(* Logix 5000 project; controller STAT 1756-L72 rev 20.12; software revision 20.04; part 27 of 34 *)
(* tags used below, declared in another part *)
   B3 : DINT[35];
   N20 : DINT[50];
   N7 : DINT[150];
   N9 : DINT[200];
   S : INT[164];
   T4 : TIMER[100];
   S_ppas_HT : DINT;
   S_ppas_l1op008 : DINT;
   S_ppas_L2op008 : DINT;
(* LANCY, continued *)

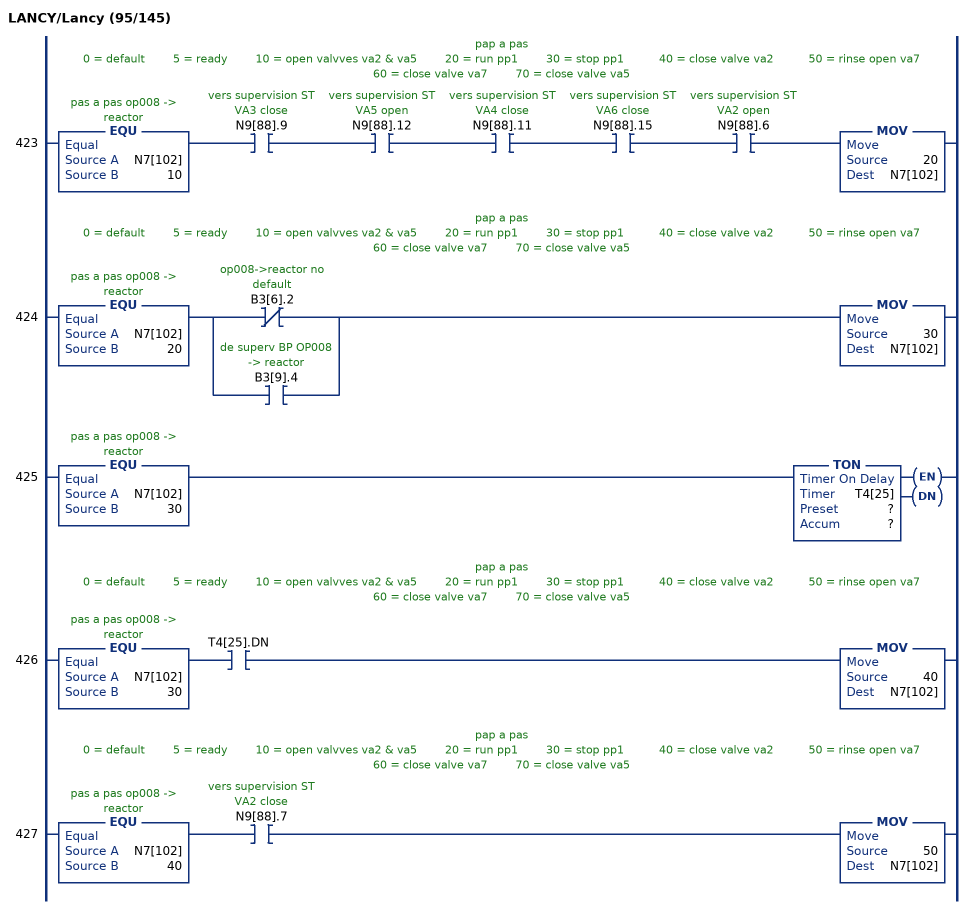
   // pap a pas
   // 0 = default        5 = ready        10 = open valvves va2 & va5        20 = run pp1        30 = stop pp1          40 = close valve va2          50 = rinse open va7            60 = close valve va7        70 = close valve va5
   423: EQU(N7[102],10)XIC(N9[88].9)XIC(N9[88].12)XIC(N9[88].11)XIC(N9[88].15)XIC(N9[88].6)MOV(20,N7[102]);
   // pap a pas
   // 0 = default        5 = ready        10 = open valvves va2 & va5        20 = run pp1        30 = stop pp1          40 = close valve va2          50 = rinse open va7            60 = close valve va7        70 = close valve va5
   424: EQU(N7[102],20)[XIO(B3[6].2) ,XIC(B3[9].4) ]MOV(30,N7[102]);
   425: EQU(N7[102],30)TON(T4[25],?,?);
   // pap a pas
   // 0 = default        5 = ready        10 = open valvves va2 & va5        20 = run pp1        30 = stop pp1          40 = close valve va2          50 = rinse open va7            60 = close valve va7        70 = close valve va5
   426: EQU(N7[102],30)XIC(T4[25].DN)MOV(40,N7[102]);
   // pap a pas
   // 0 = default        5 = ready        10 = open valvves va2 & va5        20 = run pp1        30 = stop pp1          40 = close valve va2          50 = rinse open va7            60 = close valve va7        70 = close valve va5
   427: EQU(N7[102],40)XIC(N9[88].7)MOV(50,N7[102]);
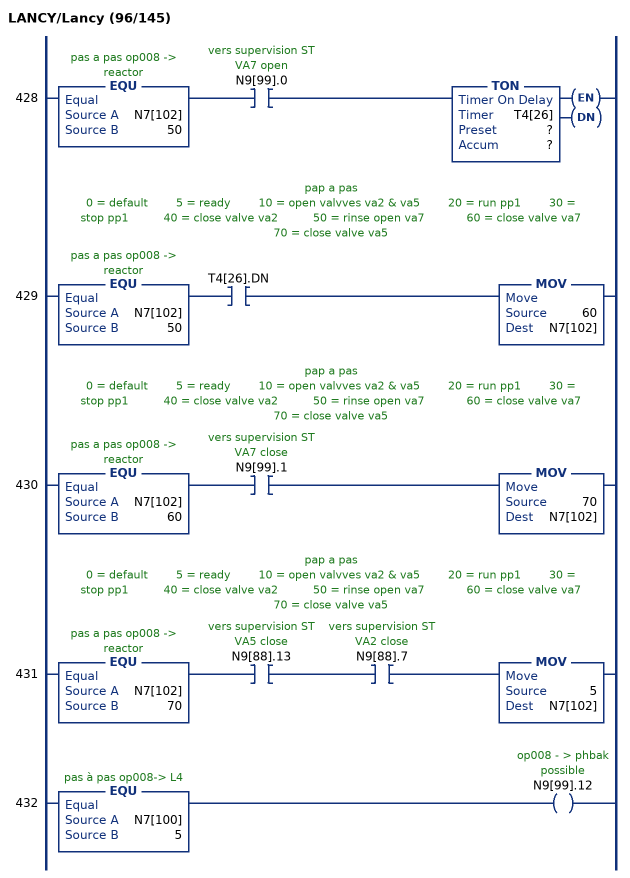
   428: EQU(N7[102],50)XIC(N9[99].0)TON(T4[26],?,?);
   // pap a pas
   // 0 = default        5 = ready        10 = open valvves va2 & va5        20 = run pp1        30 = stop pp1          40 = close valve va2          50 = rinse open va7            60 = close valve va7        70 = close valve va5
   429: EQU(N7[102],50)XIC(T4[26].DN)MOV(60,N7[102]);
   // pap a pas
   // 0 = default        5 = ready        10 = open valvves va2 & va5        20 = run pp1        30 = stop pp1          40 = close valve va2          50 = rinse open va7            60 = close valve va7        70 = close valve va5
   430: EQU(N7[102],60)XIC(N9[99].1)MOV(70,N7[102]);
   // pap a pas
   // 0 = default        5 = ready        10 = open valvves va2 & va5        20 = run pp1        30 = stop pp1          40 = close valve va2          50 = rinse open va7            60 = close valve va7        70 = close valve va5
   431: EQU(N7[102],70)XIC(N9[88].13)XIC(N9[88].7)MOV(5,N7[102]);
   432: EQU(N7[100],5)OTE(N9[99].12);
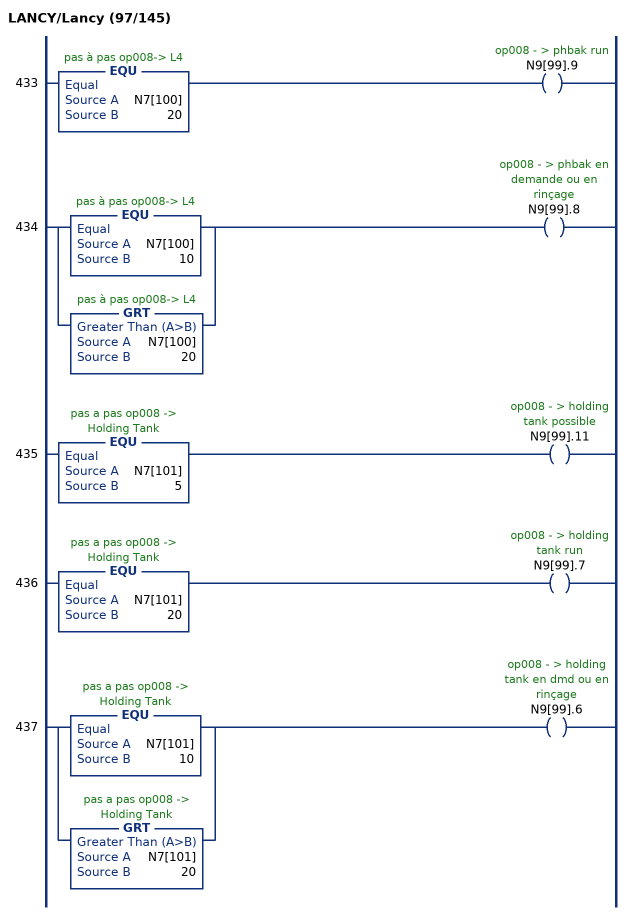
   433: EQU(N7[100],20)OTE(N9[99].9);
   434: [EQU(N7[100],10) ,GRT(N7[100],20) ]OTE(N9[99].8);
   435: EQU(N7[101],5)OTE(N9[99].11);
   436: EQU(N7[101],20)OTE(N9[99].7);
   437: [EQU(N7[101],10) ,GRT(N7[101],20) ]OTE(N9[99].6);
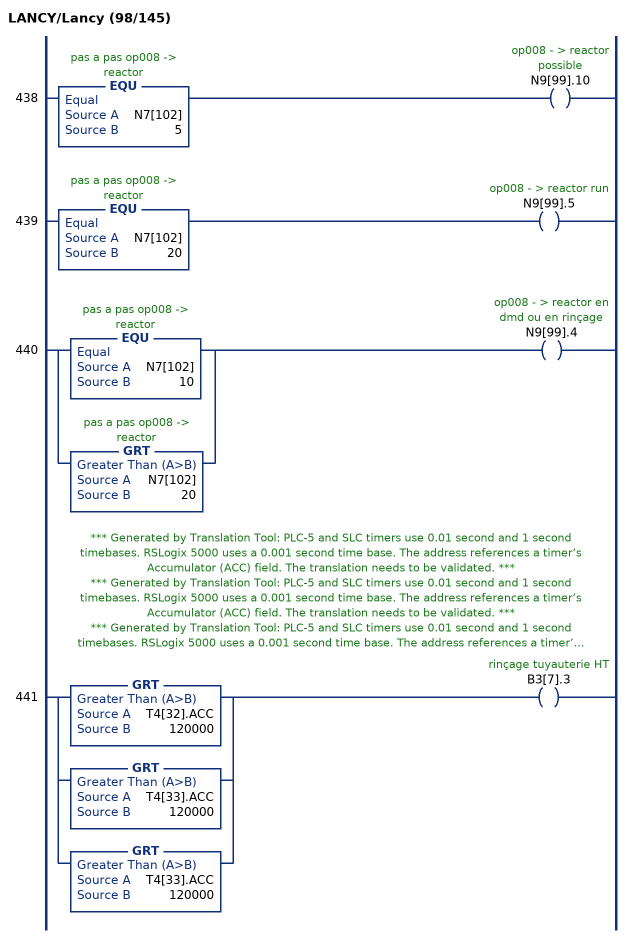
   438: EQU(N7[102],5)OTE(N9[99].10);
   439: EQU(N7[102],20)OTE(N9[99].5);
   440: [EQU(N7[102],10) ,GRT(N7[102],20) ]OTE(N9[99].4);
   // *** Generated by Translation Tool: PLC-5 and SLC timers use 0.01 second and 1 second timebases. RSLogix 5000 uses a 0.001 second time base. The address references a timer’s Accumulator (ACC) field. The translation needs to be validated. ***
   // *** Generated by Translation Tool: PLC-5 and SLC timers use 0.01 second and 1 second timebases. RSLogix 5000 uses a 0.001 second time base. The address references a timer’s Accumulator (ACC) field. The translation needs to be validated. ***
   // *** Generated by Translation Tool: PLC-5 and SLC timers use 0.01 second and 1 second timebases. RSLogix 5000 uses a 0.001 second time base. The address references a timer’s Accumulator (ACC) field. The translation needs to be validated. ***
   441: [GRT(T4[32].ACC,120000) ,GRT(T4[33].ACC,120000) ,GRT(T4[33].ACC,120000) ]OTE(B3[7].3);
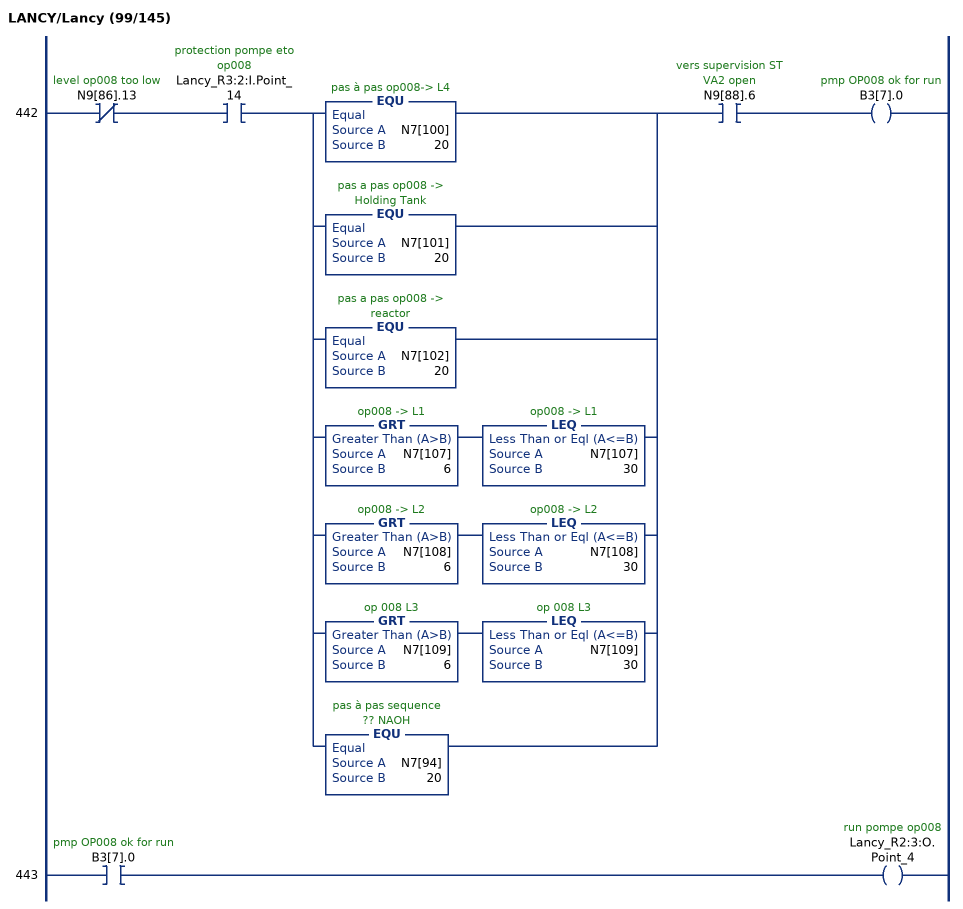
   442: XIO(N9[86].13)XIC(Lancy_R3:2:I.Point_14)[EQU(N7[100],20) ,EQU(N7[101],20) ,EQU(N7[102],20) ,GRT(N7[107],6) LEQ(N7[107],30) ,GRT(N7[108],6) LEQ(N7[108],30) ,GRT(N7[109],6) LEQ(N7[109],30) ,EQU(N7[94],20) ]XIC(N9[88].6)OTE(B3[7].0);
   443: XIC(B3[7].0)OTE(Lancy_R2:3:O.Point_4);
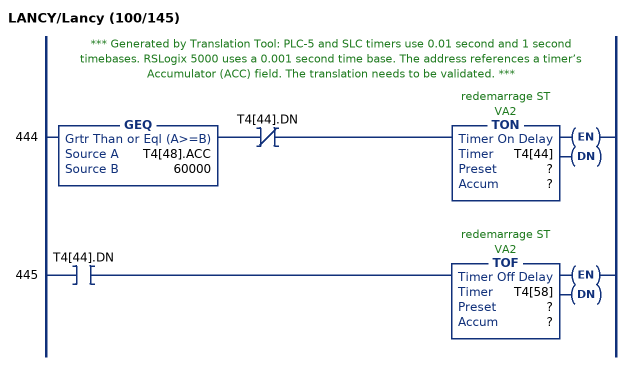
   // *** Generated by Translation Tool: PLC-5 and SLC timers use 0.01 second and 1 second timebases. RSLogix 5000 uses a 0.001 second time base. The address references a timer’s Accumulator (ACC) field. The translation needs to be validated. ***
   444: GEQ(T4[48].ACC,60000)XIO(T4[44].DN)TON(T4[44],?,?);
   445: XIC(T4[44].DN)TOF(T4[58],?,?);
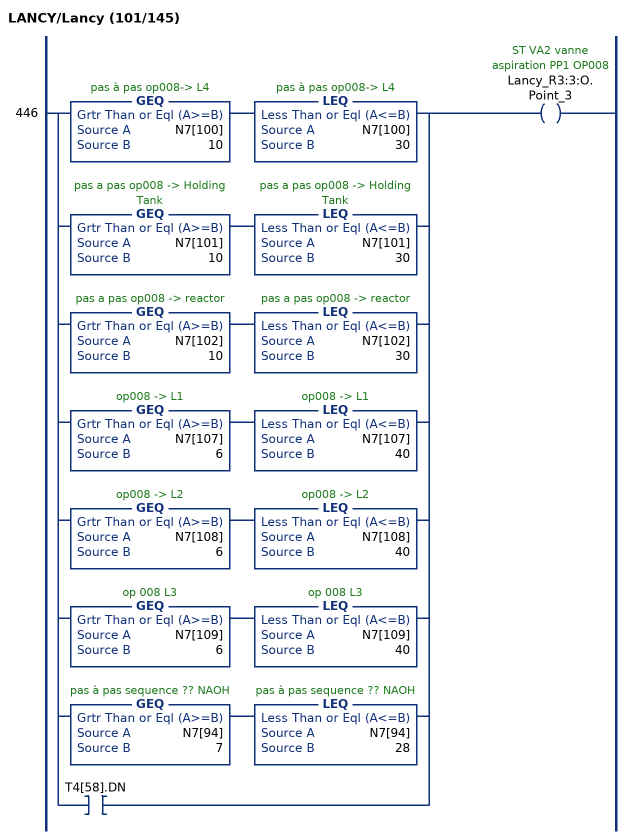
   446: [GEQ(N7[100],10) LEQ(N7[100],30) ,GEQ(N7[101],10) LEQ(N7[101],30) ,GEQ(N7[102],10) LEQ(N7[102],30) ,GEQ(N7[107],6) LEQ(N7[107],40) ,GEQ(N7[108],6) LEQ(N7[108],40) ,GEQ(N7[109],6) LEQ(N7[109],40) ,GEQ(N7[94],7) LEQ(N7[94],28) ,XIC(T4[58].DN) ]OTE(Lancy_R3:3:O.Point_3);
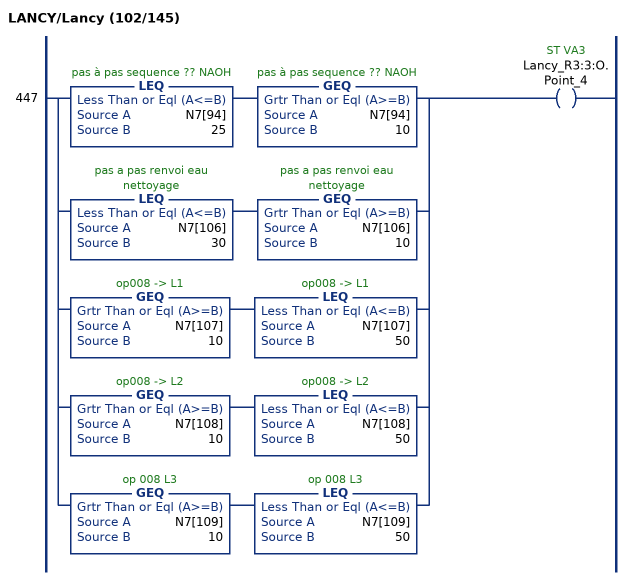
   447: [LEQ(N7[94],25) GEQ(N7[94],10) ,LEQ(N7[106],30) GEQ(N7[106],10) ,GEQ(N7[107],10) LEQ(N7[107],50) ,GEQ(N7[108],10) LEQ(N7[108],50) ,GEQ(N7[109],10) LEQ(N7[109],50) ]OTE(Lancy_R3:3:O.Point_4);
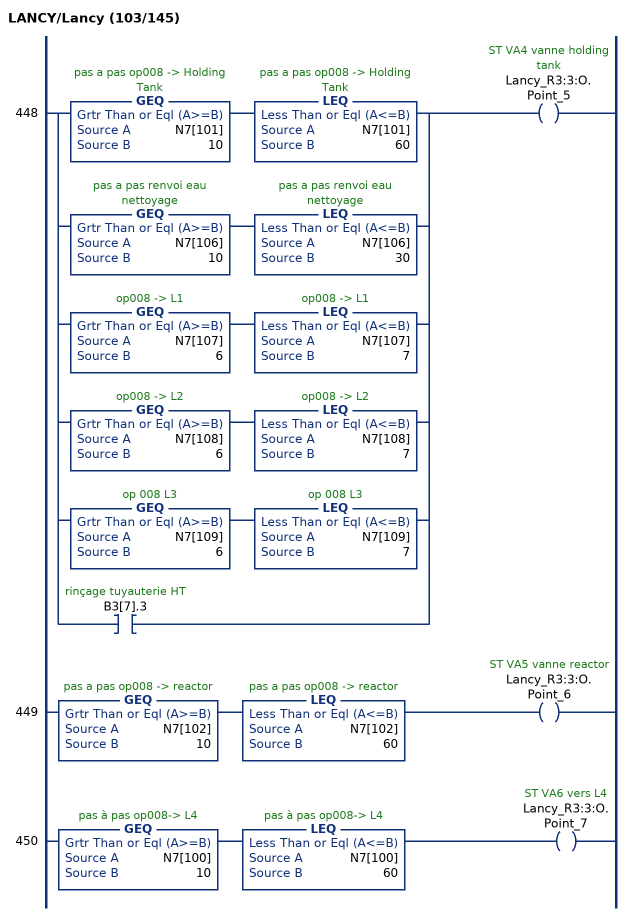
   448: [GEQ(N7[101],10) LEQ(N7[101],60) ,GEQ(N7[106],10) LEQ(N7[106],30) ,GEQ(N7[107],6) LEQ(N7[107],7) ,GEQ(N7[108],6) LEQ(N7[108],7) ,GEQ(N7[109],6) LEQ(N7[109],7) ,XIC(B3[7].3) ]OTE(Lancy_R3:3:O.Point_5);
   449: GEQ(N7[102],10)LEQ(N7[102],60)OTE(Lancy_R3:3:O.Point_6);
   450: GEQ(N7[100],10)LEQ(N7[100],60)OTE(Lancy_R3:3:O.Point_7);
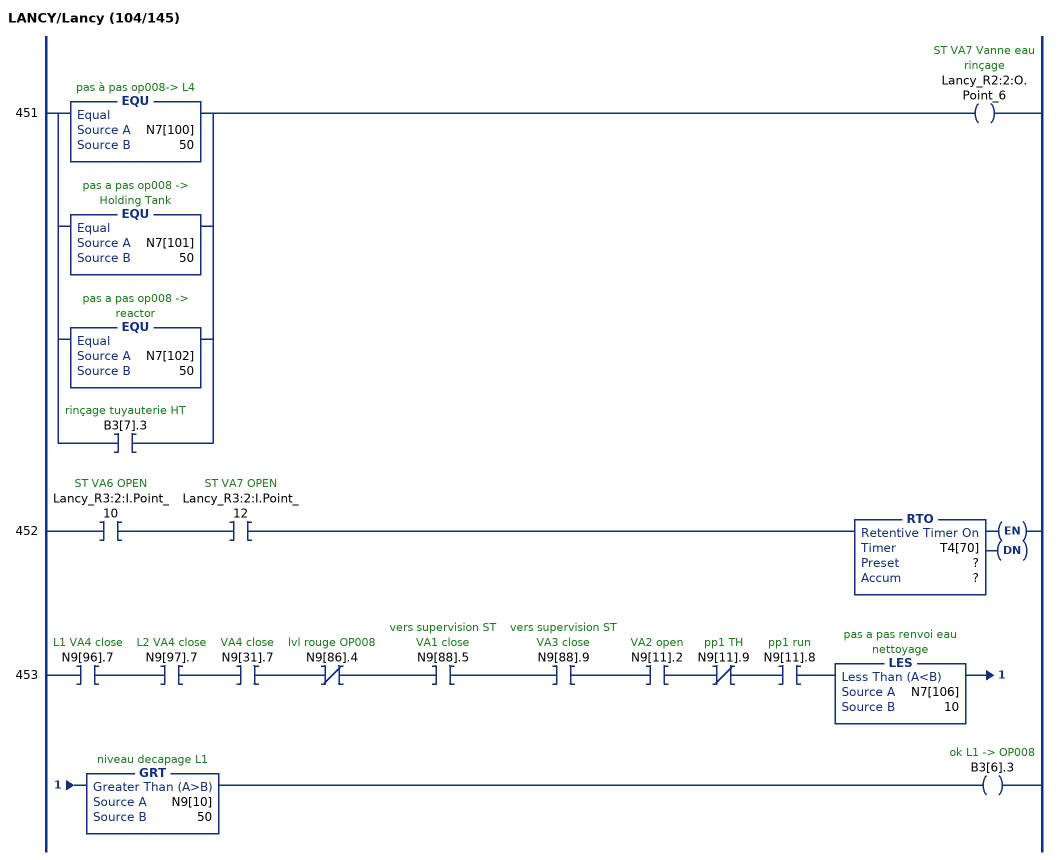
   451: [EQU(N7[100],50) ,EQU(N7[101],50) ,EQU(N7[102],50) ,XIC(B3[7].3) ]OTE(Lancy_R2:2:O.Point_6);
   452: XIC(Lancy_R3:2:I.Point_10)XIC(Lancy_R3:2:I.Point_12)RTO(T4[70],?,?);
   453: XIC(N9[96].7)XIC(N9[97].7)XIC(N9[31].7)XIO(N9[86].4)XIC(N9[88].5)XIC(N9[88].9)XIC(N9[11].2)XIO(N9[11].9)XIC(N9[11].8)LES(N7[106],10)GRT(N9[10],50)OTE(B3[6].3);
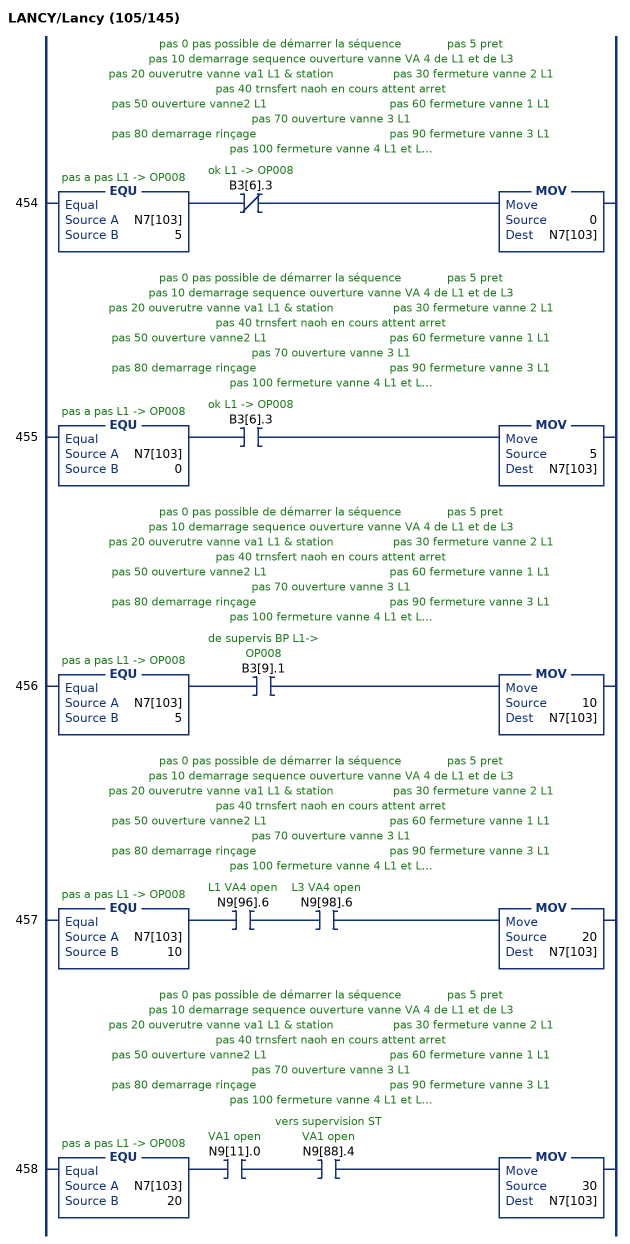
   // pas 0 pas possible de démarrer la séquence             pas 5 pret                                                 pas 10 demarrage sequence ouverture vanne VA 4 de L1 et de L3
   // pas 20 ouverutre vanne va1 L1 & station                 pas 30 fermeture vanne 2 L1                       pas 40 trnsfert naoh en cours attent arret
   // pas 50 ouverture vanne2 L1                                   pas 60 fermeture vanne 1 L1                       pas 70 ouverture vanne 3 L1
   // pas 80 demarrage rinçage                                      pas 90 fermeture vanne 3 L1                       pas 100 fermeture vanne 4 L1 et L3
   // pas 110 fermeture vanne station 1
   454: EQU(N7[103],5)XIO(B3[6].3)MOV(0,N7[103]);
   // pas 0 pas possible de démarrer la séquence             pas 5 pret                                                 pas 10 demarrage sequence ouverture vanne VA 4 de L1 et de L3
   // pas 20 ouverutre vanne va1 L1 & station                 pas 30 fermeture vanne 2 L1                       pas 40 trnsfert naoh en cours attent arret
   // pas 50 ouverture vanne2 L1                                   pas 60 fermeture vanne 1 L1                       pas 70 ouverture vanne 3 L1
   // pas 80 demarrage rinçage                                      pas 90 fermeture vanne 3 L1                       pas 100 fermeture vanne 4 L1 et L3
   // pas 110 fermeture vanne station 1
   455: EQU(N7[103],0)XIC(B3[6].3)MOV(5,N7[103]);
   // pas 0 pas possible de démarrer la séquence             pas 5 pret                                                 pas 10 demarrage sequence ouverture vanne VA 4 de L1 et de L3
   // pas 20 ouverutre vanne va1 L1 & station                 pas 30 fermeture vanne 2 L1                       pas 40 trnsfert naoh en cours attent arret
   // pas 50 ouverture vanne2 L1                                   pas 60 fermeture vanne 1 L1                       pas 70 ouverture vanne 3 L1
   // pas 80 demarrage rinçage                                      pas 90 fermeture vanne 3 L1                       pas 100 fermeture vanne 4 L1 et L3
   // pas 110 fermeture vanne station 1
   456: EQU(N7[103],5)XIC(B3[9].1)MOV(10,N7[103]);
   // pas 0 pas possible de démarrer la séquence             pas 5 pret                                                 pas 10 demarrage sequence ouverture vanne VA 4 de L1 et de L3
   // pas 20 ouverutre vanne va1 L1 & station                 pas 30 fermeture vanne 2 L1                       pas 40 trnsfert naoh en cours attent arret
   // pas 50 ouverture vanne2 L1                                   pas 60 fermeture vanne 1 L1                       pas 70 ouverture vanne 3 L1
   // pas 80 demarrage rinçage                                      pas 90 fermeture vanne 3 L1                       pas 100 fermeture vanne 4 L1 et L3
   // pas 110 fermeture vanne station 1
   457: EQU(N7[103],10)XIC(N9[96].6)XIC(N9[98].6)MOV(20,N7[103]);
   // pas 0 pas possible de démarrer la séquence             pas 5 pret                                                 pas 10 demarrage sequence ouverture vanne VA 4 de L1 et de L3
   // pas 20 ouverutre vanne va1 L1 & station                 pas 30 fermeture vanne 2 L1                       pas 40 trnsfert naoh en cours attent arret
   // pas 50 ouverture vanne2 L1                                   pas 60 fermeture vanne 1 L1                       pas 70 ouverture vanne 3 L1
   // pas 80 demarrage rinçage                                      pas 90 fermeture vanne 3 L1                       pas 100 fermeture vanne 4 L1 et L3
   // pas 110 fermeture vanne station 1
   458: EQU(N7[103],20)XIC(N9[11].0)XIC(N9[88].4)MOV(30,N7[103]);
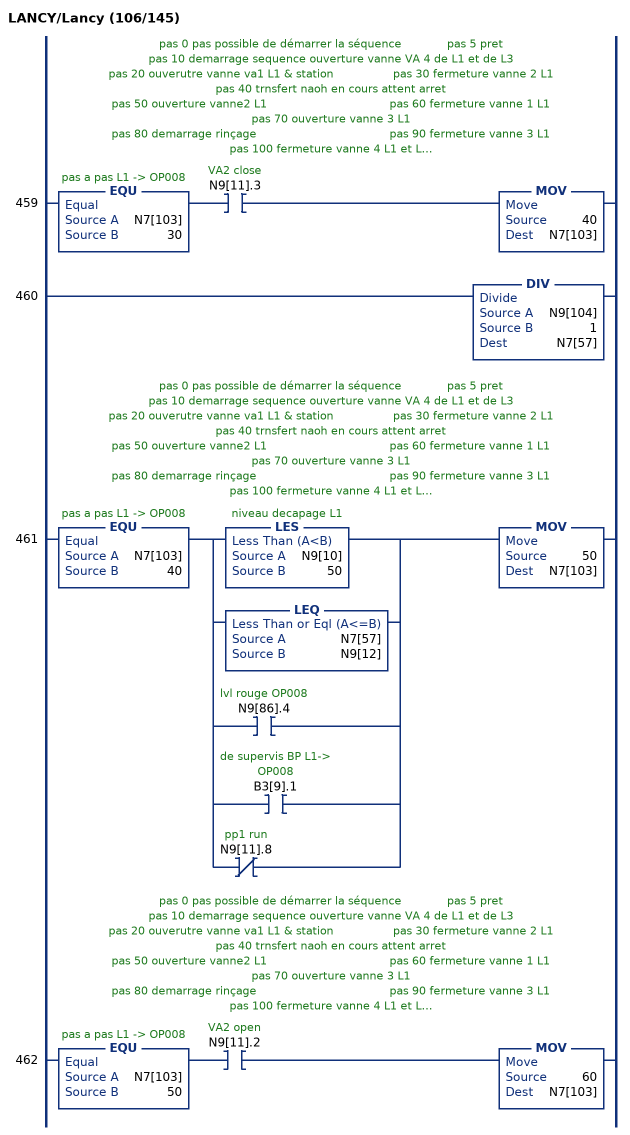
   // pas 0 pas possible de démarrer la séquence             pas 5 pret                                                 pas 10 demarrage sequence ouverture vanne VA 4 de L1 et de L3
   // pas 20 ouverutre vanne va1 L1 & station                 pas 30 fermeture vanne 2 L1                       pas 40 trnsfert naoh en cours attent arret
   // pas 50 ouverture vanne2 L1                                   pas 60 fermeture vanne 1 L1                       pas 70 ouverture vanne 3 L1
   // pas 80 demarrage rinçage                                      pas 90 fermeture vanne 3 L1                       pas 100 fermeture vanne 4 L1 et L3
   // pas 110 fermeture vanne station 1
   459: EQU(N7[103],30)XIC(N9[11].3)MOV(40,N7[103]);
   460: DIV(N9[104],1,N7[57]);
   // pas 0 pas possible de démarrer la séquence             pas 5 pret                                                 pas 10 demarrage sequence ouverture vanne VA 4 de L1 et de L3
   // pas 20 ouverutre vanne va1 L1 & station                 pas 30 fermeture vanne 2 L1                       pas 40 trnsfert naoh en cours attent arret
   // pas 50 ouverture vanne2 L1                                   pas 60 fermeture vanne 1 L1                       pas 70 ouverture vanne 3 L1
   // pas 80 demarrage rinçage                                      pas 90 fermeture vanne 3 L1                       pas 100 fermeture vanne 4 L1 et L3
   // pas 110 fermeture vanne station 1
   461: EQU(N7[103],40)[LES(N9[10],50) ,LEQ(N7[57],N9[12]) ,XIC(N9[86].4) ,XIC(B3[9].1) ,XIO(N9[11].8) ]MOV(50,N7[103]);
   // pas 0 pas possible de démarrer la séquence             pas 5 pret                                                 pas 10 demarrage sequence ouverture vanne VA 4 de L1 et de L3
   // pas 20 ouverutre vanne va1 L1 & station                 pas 30 fermeture vanne 2 L1                       pas 40 trnsfert naoh en cours attent arret
   // pas 50 ouverture vanne2 L1                                   pas 60 fermeture vanne 1 L1                       pas 70 ouverture vanne 3 L1
   // pas 80 demarrage rinçage                                      pas 90 fermeture vanne 3 L1                       pas 100 fermeture vanne 4 L1 et L3
   // pas 110 fermeture vanne station 1
   462: EQU(N7[103],50)XIC(N9[11].2)MOV(60,N7[103]);
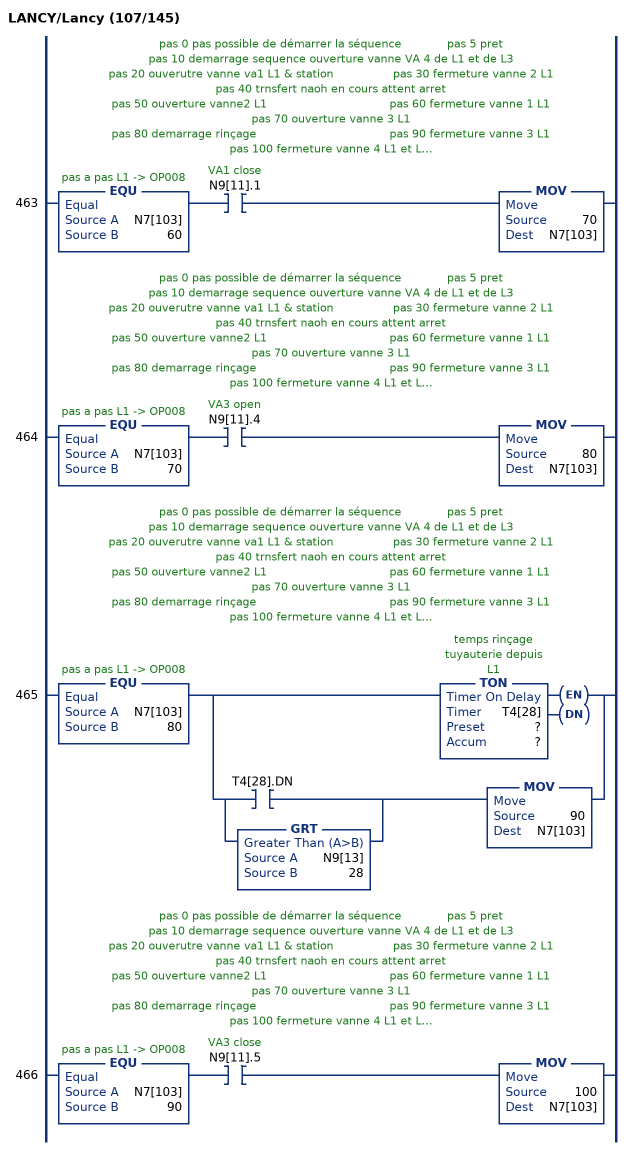
   // pas 0 pas possible de démarrer la séquence             pas 5 pret                                                 pas 10 demarrage sequence ouverture vanne VA 4 de L1 et de L3
   // pas 20 ouverutre vanne va1 L1 & station                 pas 30 fermeture vanne 2 L1                       pas 40 trnsfert naoh en cours attent arret
   // pas 50 ouverture vanne2 L1                                   pas 60 fermeture vanne 1 L1                       pas 70 ouverture vanne 3 L1
   // pas 80 demarrage rinçage                                      pas 90 fermeture vanne 3 L1                       pas 100 fermeture vanne 4 L1 et L3
   // pas 110 fermeture vanne station 1
   463: EQU(N7[103],60)XIC(N9[11].1)MOV(70,N7[103]);
   // pas 0 pas possible de démarrer la séquence             pas 5 pret                                                 pas 10 demarrage sequence ouverture vanne VA 4 de L1 et de L3
   // pas 20 ouverutre vanne va1 L1 & station                 pas 30 fermeture vanne 2 L1                       pas 40 trnsfert naoh en cours attent arret
   // pas 50 ouverture vanne2 L1                                   pas 60 fermeture vanne 1 L1                       pas 70 ouverture vanne 3 L1
   // pas 80 demarrage rinçage                                      pas 90 fermeture vanne 3 L1                       pas 100 fermeture vanne 4 L1 et L3
   // pas 110 fermeture vanne station 1
   464: EQU(N7[103],70)XIC(N9[11].4)MOV(80,N7[103]);
   // pas 0 pas possible de démarrer la séquence             pas 5 pret                                                 pas 10 demarrage sequence ouverture vanne VA 4 de L1 et de L3
   // pas 20 ouverutre vanne va1 L1 & station                 pas 30 fermeture vanne 2 L1                       pas 40 trnsfert naoh en cours attent arret
   // pas 50 ouverture vanne2 L1                                   pas 60 fermeture vanne 1 L1                       pas 70 ouverture vanne 3 L1
   // pas 80 demarrage rinçage                                      pas 90 fermeture vanne 3 L1                       pas 100 fermeture vanne 4 L1 et L3
   // pas 110 fermeture vanne station 1
   465: EQU(N7[103],80)[TON(T4[28],?,?) ,[XIC(T4[28].DN) ,GRT(N9[13],28) ] MOV(90,N7[103]) ];
   // pas 0 pas possible de démarrer la séquence             pas 5 pret                                                 pas 10 demarrage sequence ouverture vanne VA 4 de L1 et de L3
   // pas 20 ouverutre vanne va1 L1 & station                 pas 30 fermeture vanne 2 L1                       pas 40 trnsfert naoh en cours attent arret
   // pas 50 ouverture vanne2 L1                                   pas 60 fermeture vanne 1 L1                       pas 70 ouverture vanne 3 L1
   // pas 80 demarrage rinçage                                      pas 90 fermeture vanne 3 L1                       pas 100 fermeture vanne 4 L1 et L3
   // pas 110 fermeture vanne station 1
   466: EQU(N7[103],90)XIC(N9[11].5)MOV(100,N7[103]);
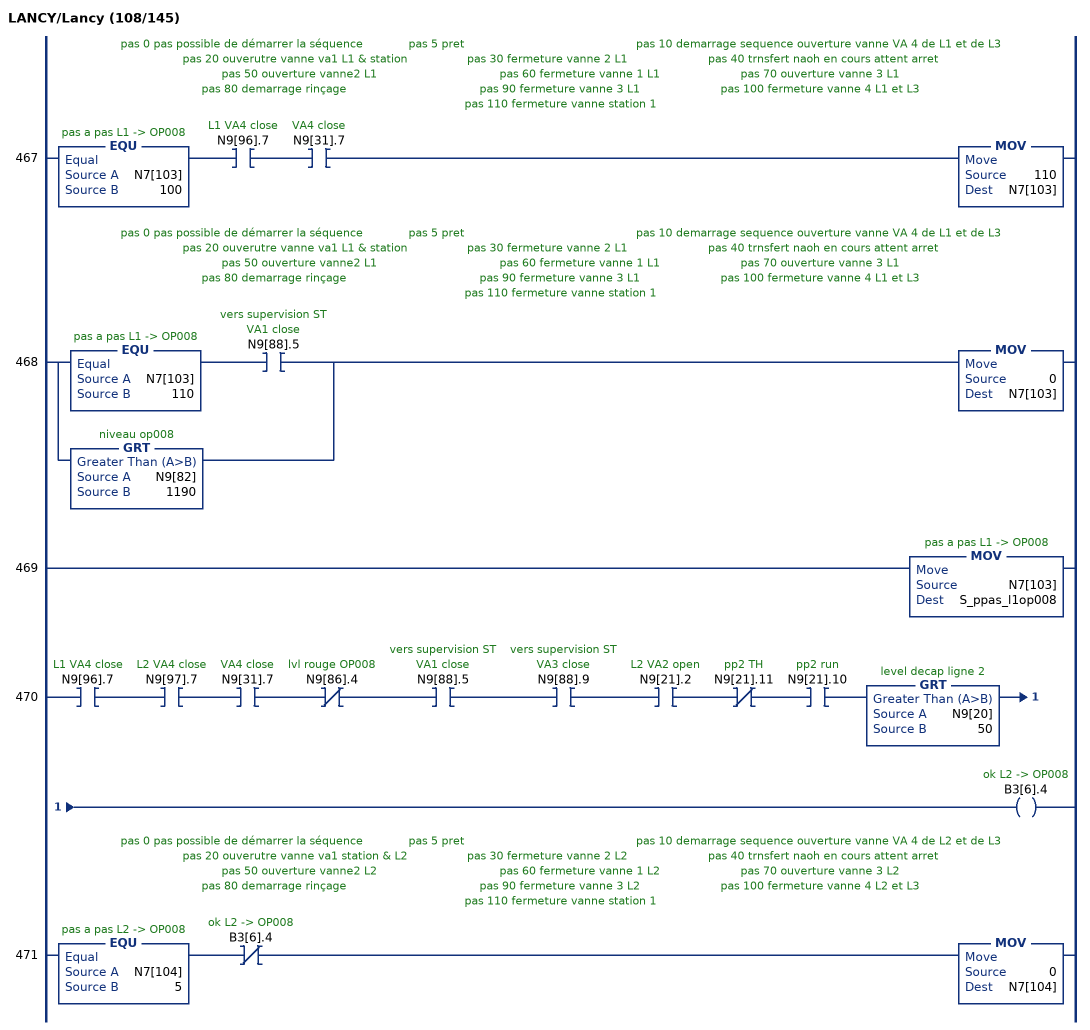
   // pas 0 pas possible de démarrer la séquence             pas 5 pret                                                 pas 10 demarrage sequence ouverture vanne VA 4 de L1 et de L3
   // pas 20 ouverutre vanne va1 L1 & station                 pas 30 fermeture vanne 2 L1                       pas 40 trnsfert naoh en cours attent arret
   // pas 50 ouverture vanne2 L1                                   pas 60 fermeture vanne 1 L1                       pas 70 ouverture vanne 3 L1
   // pas 80 demarrage rinçage                                      pas 90 fermeture vanne 3 L1                       pas 100 fermeture vanne 4 L1 et L3
   // pas 110 fermeture vanne station 1
   467: EQU(N7[103],100)XIC(N9[96].7)XIC(N9[31].7)MOV(110,N7[103]);
   // pas 0 pas possible de démarrer la séquence             pas 5 pret                                                 pas 10 demarrage sequence ouverture vanne VA 4 de L1 et de L3
   // pas 20 ouverutre vanne va1 L1 & station                 pas 30 fermeture vanne 2 L1                       pas 40 trnsfert naoh en cours attent arret
   // pas 50 ouverture vanne2 L1                                   pas 60 fermeture vanne 1 L1                       pas 70 ouverture vanne 3 L1
   // pas 80 demarrage rinçage                                      pas 90 fermeture vanne 3 L1                       pas 100 fermeture vanne 4 L1 et L3
   // pas 110 fermeture vanne station 1
   468: [EQU(N7[103],110) XIC(N9[88].5) ,GRT(N9[82],1190) ]MOV(0,N7[103]);
   469: MOV(N7[103],S_ppas_l1op008);
   470: XIC(N9[96].7)XIC(N9[97].7)XIC(N9[31].7)XIO(N9[86].4)XIC(N9[88].5)XIC(N9[88].9)XIC(N9[21].2)XIO(N9[21].11)XIC(N9[21].10)GRT(N9[20],50)OTE(B3[6].4);
   // pas 0 pas possible de démarrer la séquence             pas 5 pret                                                 pas 10 demarrage sequence ouverture vanne VA 4 de L2 et de L3
   // pas 20 ouverutre vanne va1 station & L2                 pas 30 fermeture vanne 2 L2                       pas 40 trnsfert naoh en cours attent arret
   // pas 50 ouverture vanne2 L2                                   pas 60 fermeture vanne 1 L2                       pas 70 ouverture vanne 3 L2
   // pas 80 demarrage rinçage                                      pas 90 fermeture vanne 3 L2                       pas 100 fermeture vanne 4 L2 et L3
   // pas 110 fermeture vanne station 1
   471: EQU(N7[104],5)XIO(B3[6].4)MOV(0,N7[104]);
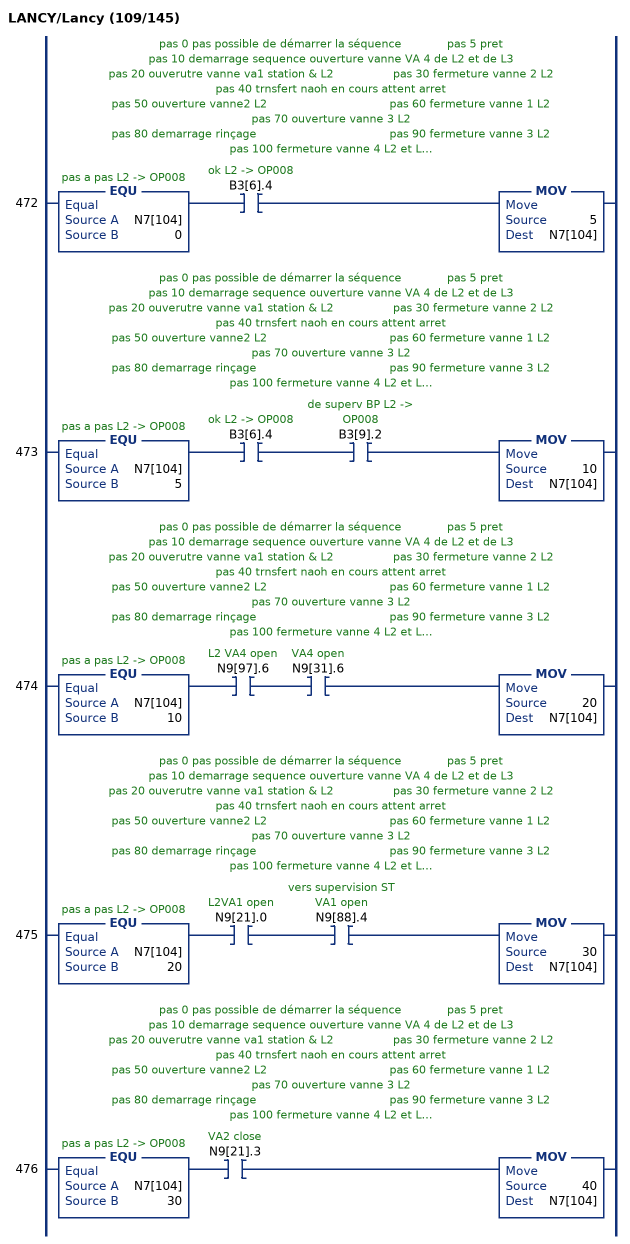
   // pas 0 pas possible de démarrer la séquence             pas 5 pret                                                 pas 10 demarrage sequence ouverture vanne VA 4 de L2 et de L3
   // pas 20 ouverutre vanne va1 station & L2                 pas 30 fermeture vanne 2 L2                       pas 40 trnsfert naoh en cours attent arret
   // pas 50 ouverture vanne2 L2                                   pas 60 fermeture vanne 1 L2                       pas 70 ouverture vanne 3 L2
   // pas 80 demarrage rinçage                                      pas 90 fermeture vanne 3 L2                       pas 100 fermeture vanne 4 L2 et L3
   // pas 110 fermeture vanne station 1
   472: EQU(N7[104],0)XIC(B3[6].4)MOV(5,N7[104]);
   // pas 0 pas possible de démarrer la séquence             pas 5 pret                                                 pas 10 demarrage sequence ouverture vanne VA 4 de L2 et de L3
   // pas 20 ouverutre vanne va1 station & L2                 pas 30 fermeture vanne 2 L2                       pas 40 trnsfert naoh en cours attent arret
   // pas 50 ouverture vanne2 L2                                   pas 60 fermeture vanne 1 L2                       pas 70 ouverture vanne 3 L2
   // pas 80 demarrage rinçage                                      pas 90 fermeture vanne 3 L2                       pas 100 fermeture vanne 4 L2 et L3
   // pas 110 fermeture vanne station 1
   473: EQU(N7[104],5)XIC(B3[6].4)XIC(B3[9].2)MOV(10,N7[104]);
   // pas 0 pas possible de démarrer la séquence             pas 5 pret                                                 pas 10 demarrage sequence ouverture vanne VA 4 de L2 et de L3
   // pas 20 ouverutre vanne va1 station & L2                 pas 30 fermeture vanne 2 L2                       pas 40 trnsfert naoh en cours attent arret
   // pas 50 ouverture vanne2 L2                                   pas 60 fermeture vanne 1 L2                       pas 70 ouverture vanne 3 L2
   // pas 80 demarrage rinçage                                      pas 90 fermeture vanne 3 L2                       pas 100 fermeture vanne 4 L2 et L3
   // pas 110 fermeture vanne station 1
   474: EQU(N7[104],10)XIC(N9[97].6)XIC(N9[31].6)MOV(20,N7[104]);
   // pas 0 pas possible de démarrer la séquence             pas 5 pret                                                 pas 10 demarrage sequence ouverture vanne VA 4 de L2 et de L3
   // pas 20 ouverutre vanne va1 station & L2                 pas 30 fermeture vanne 2 L2                       pas 40 trnsfert naoh en cours attent arret
   // pas 50 ouverture vanne2 L2                                   pas 60 fermeture vanne 1 L2                       pas 70 ouverture vanne 3 L2
   // pas 80 demarrage rinçage                                      pas 90 fermeture vanne 3 L2                       pas 100 fermeture vanne 4 L2 et L3
   // pas 110 fermeture vanne station 1
   475: EQU(N7[104],20)XIC(N9[21].0)XIC(N9[88].4)MOV(30,N7[104]);
   // pas 0 pas possible de démarrer la séquence             pas 5 pret                                                 pas 10 demarrage sequence ouverture vanne VA 4 de L2 et de L3
   // pas 20 ouverutre vanne va1 station & L2                 pas 30 fermeture vanne 2 L2                       pas 40 trnsfert naoh en cours attent arret
   // pas 50 ouverture vanne2 L2                                   pas 60 fermeture vanne 1 L2                       pas 70 ouverture vanne 3 L2
   // pas 80 demarrage rinçage                                      pas 90 fermeture vanne 3 L2                       pas 100 fermeture vanne 4 L2 et L3
   // pas 110 fermeture vanne station 1
   476: EQU(N7[104],30)XIC(N9[21].3)MOV(40,N7[104]);
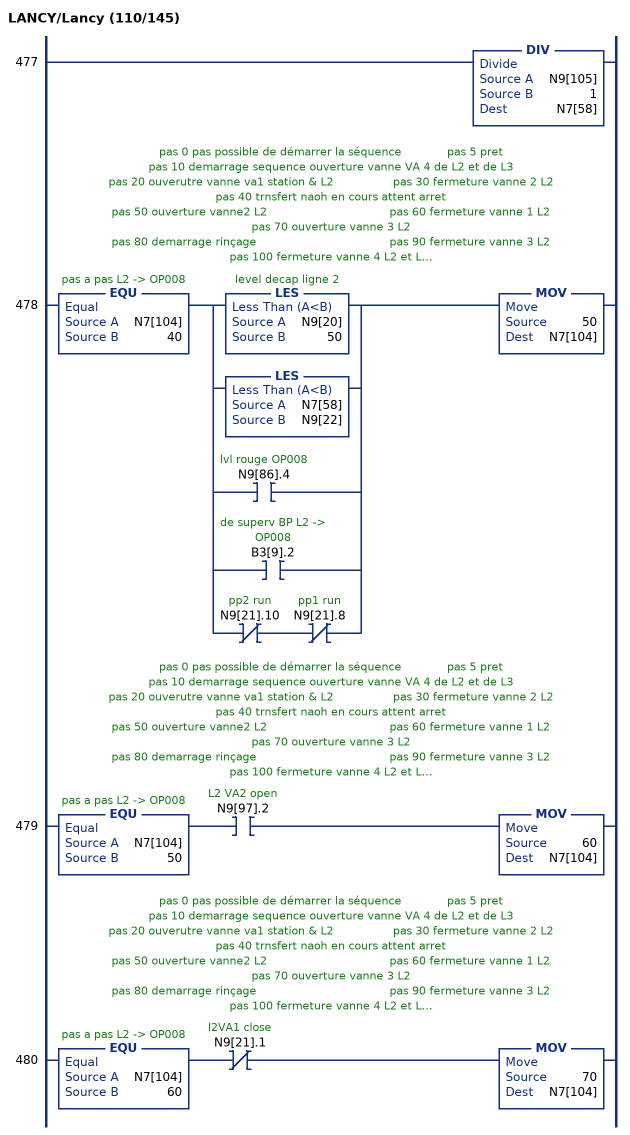
   477: DIV(N9[105],1,N7[58]);
   // pas 0 pas possible de démarrer la séquence             pas 5 pret                                                 pas 10 demarrage sequence ouverture vanne VA 4 de L2 et de L3
   // pas 20 ouverutre vanne va1 station & L2                 pas 30 fermeture vanne 2 L2                       pas 40 trnsfert naoh en cours attent arret
   // pas 50 ouverture vanne2 L2                                   pas 60 fermeture vanne 1 L2                       pas 70 ouverture vanne 3 L2
   // pas 80 demarrage rinçage                                      pas 90 fermeture vanne 3 L2                       pas 100 fermeture vanne 4 L2 et L3
   // pas 110 fermeture vanne station 1
   478: EQU(N7[104],40)[LES(N9[20],50) ,LES(N7[58],N9[22]) ,XIC(N9[86].4) ,XIC(B3[9].2) ,XIO(N9[21].10) XIO(N9[21].8) ]MOV(50,N7[104]);
   // pas 0 pas possible de démarrer la séquence             pas 5 pret                                                 pas 10 demarrage sequence ouverture vanne VA 4 de L2 et de L3
   // pas 20 ouverutre vanne va1 station & L2                 pas 30 fermeture vanne 2 L2                       pas 40 trnsfert naoh en cours attent arret
   // pas 50 ouverture vanne2 L2                                   pas 60 fermeture vanne 1 L2                       pas 70 ouverture vanne 3 L2
   // pas 80 demarrage rinçage                                      pas 90 fermeture vanne 3 L2                       pas 100 fermeture vanne 4 L2 et L3
   // pas 110 fermeture vanne station 1
   479: EQU(N7[104],50)XIC(N9[97].2)MOV(60,N7[104]);
   // pas 0 pas possible de démarrer la séquence             pas 5 pret                                                 pas 10 demarrage sequence ouverture vanne VA 4 de L2 et de L3
   // pas 20 ouverutre vanne va1 station & L2                 pas 30 fermeture vanne 2 L2                       pas 40 trnsfert naoh en cours attent arret
   // pas 50 ouverture vanne2 L2                                   pas 60 fermeture vanne 1 L2                       pas 70 ouverture vanne 3 L2
   // pas 80 demarrage rinçage                                      pas 90 fermeture vanne 3 L2                       pas 100 fermeture vanne 4 L2 et L3
   // pas 110 fermeture vanne station 1
   480: EQU(N7[104],60)XIO(N9[21].1)MOV(70,N7[104]);
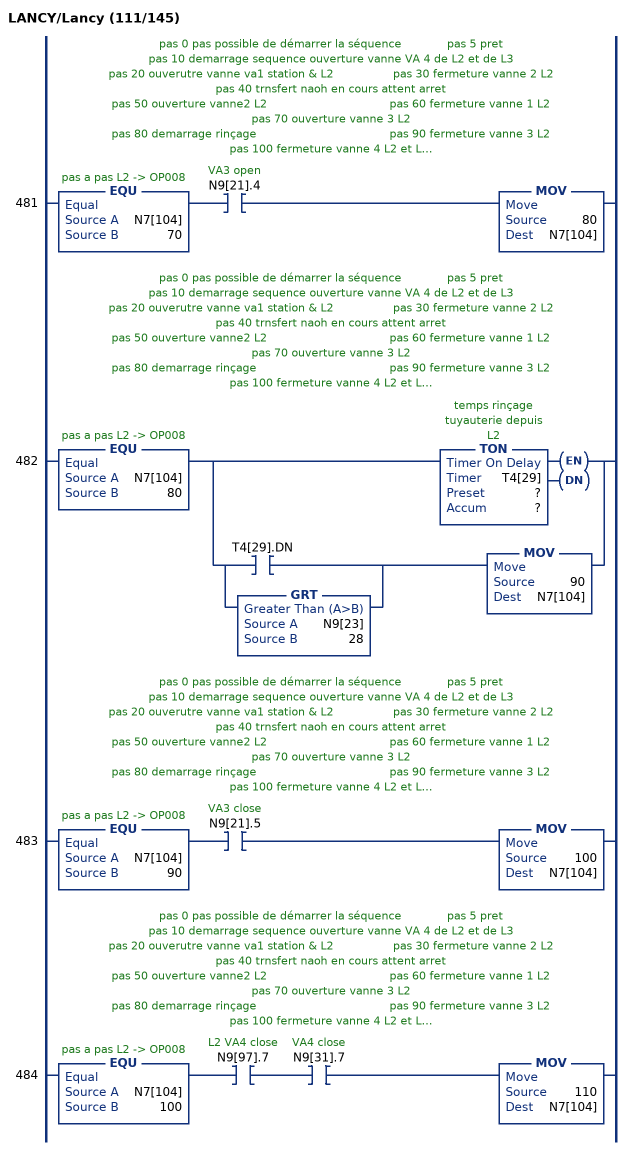
   // pas 0 pas possible de démarrer la séquence             pas 5 pret                                                 pas 10 demarrage sequence ouverture vanne VA 4 de L2 et de L3
   // pas 20 ouverutre vanne va1 station & L2                 pas 30 fermeture vanne 2 L2                       pas 40 trnsfert naoh en cours attent arret
   // pas 50 ouverture vanne2 L2                                   pas 60 fermeture vanne 1 L2                       pas 70 ouverture vanne 3 L2
   // pas 80 demarrage rinçage                                      pas 90 fermeture vanne 3 L2                       pas 100 fermeture vanne 4 L2 et L3
   // pas 110 fermeture vanne station 1
   481: EQU(N7[104],70)XIC(N9[21].4)MOV(80,N7[104]);
   // pas 0 pas possible de démarrer la séquence             pas 5 pret                                                 pas 10 demarrage sequence ouverture vanne VA 4 de L2 et de L3
   // pas 20 ouverutre vanne va1 station & L2                 pas 30 fermeture vanne 2 L2                       pas 40 trnsfert naoh en cours attent arret
   // pas 50 ouverture vanne2 L2                                   pas 60 fermeture vanne 1 L2                       pas 70 ouverture vanne 3 L2
   // pas 80 demarrage rinçage                                      pas 90 fermeture vanne 3 L2                       pas 100 fermeture vanne 4 L2 et L3
   // pas 110 fermeture vanne station 1
   482: EQU(N7[104],80)[TON(T4[29],?,?) ,[XIC(T4[29].DN) ,GRT(N9[23],28) ] MOV(90,N7[104]) ];
   // pas 0 pas possible de démarrer la séquence             pas 5 pret                                                 pas 10 demarrage sequence ouverture vanne VA 4 de L2 et de L3
   // pas 20 ouverutre vanne va1 station & L2                 pas 30 fermeture vanne 2 L2                       pas 40 trnsfert naoh en cours attent arret
   // pas 50 ouverture vanne2 L2                                   pas 60 fermeture vanne 1 L2                       pas 70 ouverture vanne 3 L2
   // pas 80 demarrage rinçage                                      pas 90 fermeture vanne 3 L2                       pas 100 fermeture vanne 4 L2 et L3
   // pas 110 fermeture vanne station 1
   483: EQU(N7[104],90)XIC(N9[21].5)MOV(100,N7[104]);
   // pas 0 pas possible de démarrer la séquence             pas 5 pret                                                 pas 10 demarrage sequence ouverture vanne VA 4 de L2 et de L3
   // pas 20 ouverutre vanne va1 station & L2                 pas 30 fermeture vanne 2 L2                       pas 40 trnsfert naoh en cours attent arret
   // pas 50 ouverture vanne2 L2                                   pas 60 fermeture vanne 1 L2                       pas 70 ouverture vanne 3 L2
   // pas 80 demarrage rinçage                                      pas 90 fermeture vanne 3 L2                       pas 100 fermeture vanne 4 L2 et L3
   // pas 110 fermeture vanne station 1
   484: EQU(N7[104],100)XIC(N9[97].7)XIC(N9[31].7)MOV(110,N7[104]);
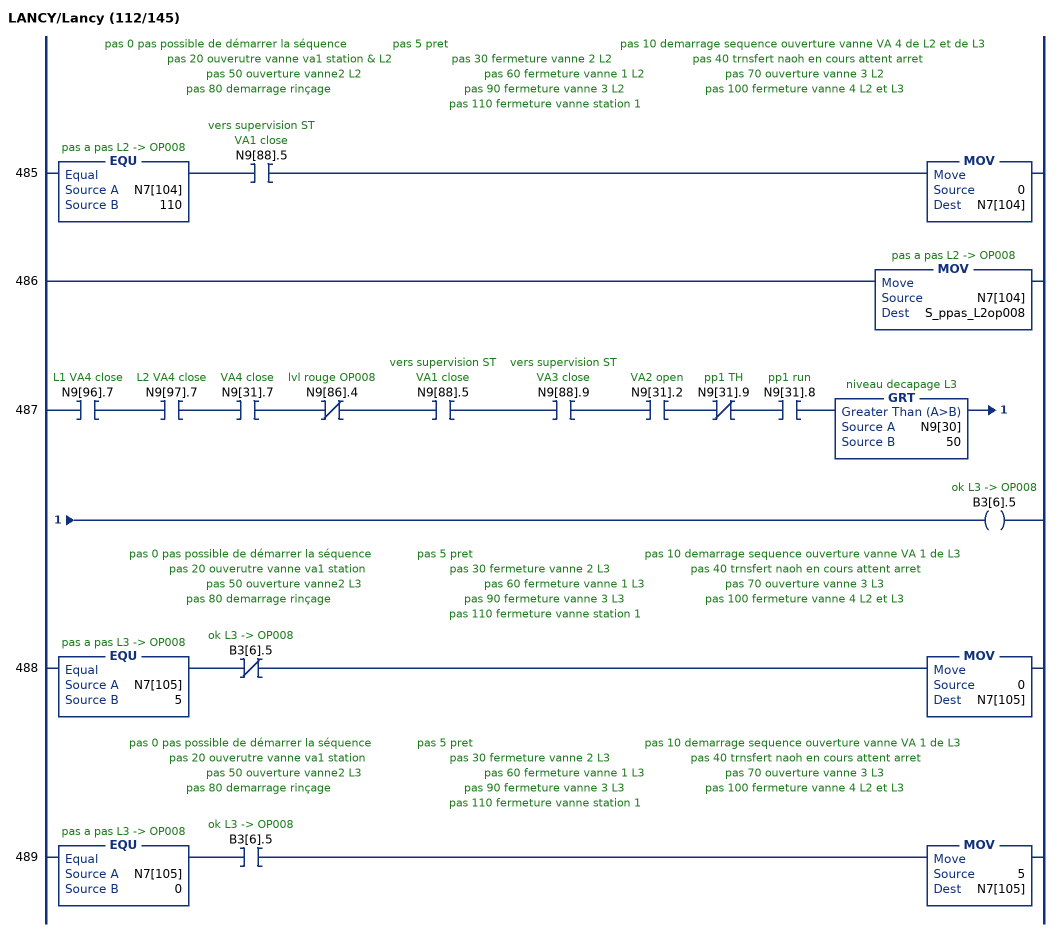
   // pas 0 pas possible de démarrer la séquence             pas 5 pret                                                 pas 10 demarrage sequence ouverture vanne VA 4 de L2 et de L3
   // pas 20 ouverutre vanne va1 station & L2                 pas 30 fermeture vanne 2 L2                       pas 40 trnsfert naoh en cours attent arret
   // pas 50 ouverture vanne2 L2                                   pas 60 fermeture vanne 1 L2                       pas 70 ouverture vanne 3 L2
   // pas 80 demarrage rinçage                                      pas 90 fermeture vanne 3 L2                       pas 100 fermeture vanne 4 L2 et L3
   // pas 110 fermeture vanne station 1
   485: EQU(N7[104],110)XIC(N9[88].5)MOV(0,N7[104]);
   486: MOV(N7[104],S_ppas_L2op008);
   487: XIC(N9[96].7)XIC(N9[97].7)XIC(N9[31].7)XIO(N9[86].4)XIC(N9[88].5)XIC(N9[88].9)XIC(N9[31].2)XIO(N9[31].9)XIC(N9[31].8)GRT(N9[30],50)OTE(B3[6].5);
   // pas 0 pas possible de démarrer la séquence             pas 5 pret                                                 pas 10 demarrage sequence ouverture vanne VA 1 de L3
   // pas 20 ouverutre vanne va1 station                        pas 30 fermeture vanne 2 L3                       pas 40 trnsfert naoh en cours attent arret
   // pas 50 ouverture vanne2 L3                                   pas 60 fermeture vanne 1 L3                       pas 70 ouverture vanne 3 L3
   // pas 80 demarrage rinçage                                      pas 90 fermeture vanne 3 L3                       pas 100 fermeture vanne 4 L2 et L3
   // pas 110 fermeture vanne station 1
   488: EQU(N7[105],5)XIO(B3[6].5)MOV(0,N7[105]);
   // pas 0 pas possible de démarrer la séquence             pas 5 pret                                                 pas 10 demarrage sequence ouverture vanne VA 1 de L3
   // pas 20 ouverutre vanne va1 station                        pas 30 fermeture vanne 2 L3                       pas 40 trnsfert naoh en cours attent arret
   // pas 50 ouverture vanne2 L3                                   pas 60 fermeture vanne 1 L3                       pas 70 ouverture vanne 3 L3
   // pas 80 demarrage rinçage                                      pas 90 fermeture vanne 3 L3                       pas 100 fermeture vanne 4 L2 et L3
   // pas 110 fermeture vanne station 1
   489: EQU(N7[105],0)XIC(B3[6].5)MOV(5,N7[105]);
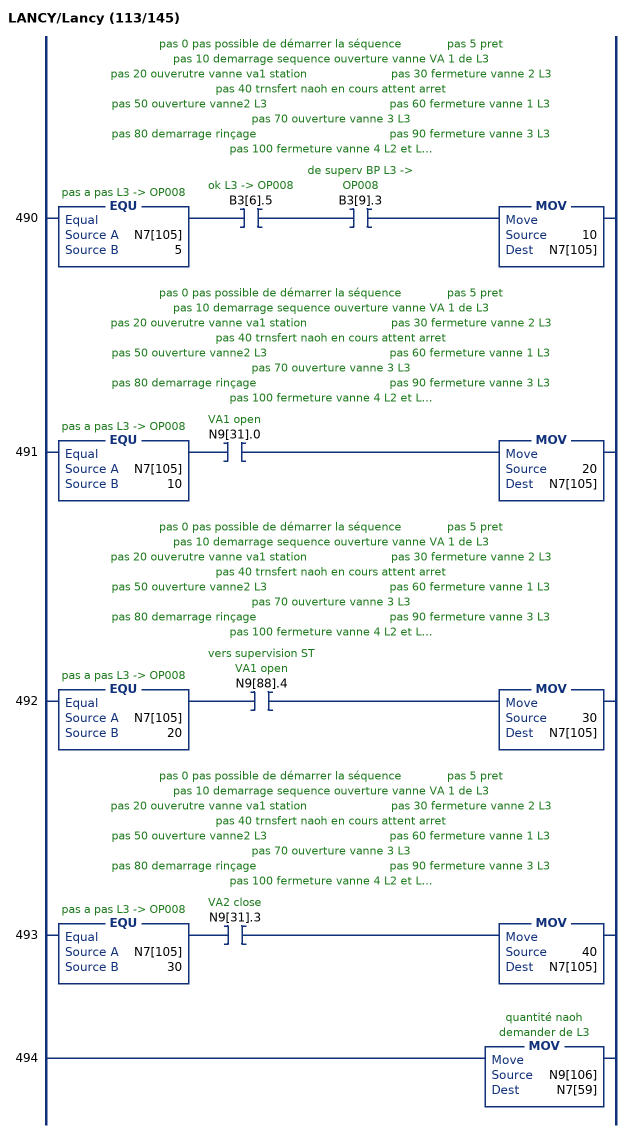
   // pas 0 pas possible de démarrer la séquence             pas 5 pret                                                 pas 10 demarrage sequence ouverture vanne VA 1 de L3
   // pas 20 ouverutre vanne va1 station                        pas 30 fermeture vanne 2 L3                       pas 40 trnsfert naoh en cours attent arret
   // pas 50 ouverture vanne2 L3                                   pas 60 fermeture vanne 1 L3                       pas 70 ouverture vanne 3 L3
   // pas 80 demarrage rinçage                                      pas 90 fermeture vanne 3 L3                       pas 100 fermeture vanne 4 L2 et L3
   // pas 110 fermeture vanne station 1
   490: EQU(N7[105],5)XIC(B3[6].5)XIC(B3[9].3)MOV(10,N7[105]);
   // pas 0 pas possible de démarrer la séquence             pas 5 pret                                                 pas 10 demarrage sequence ouverture vanne VA 1 de L3
   // pas 20 ouverutre vanne va1 station                        pas 30 fermeture vanne 2 L3                       pas 40 trnsfert naoh en cours attent arret
   // pas 50 ouverture vanne2 L3                                   pas 60 fermeture vanne 1 L3                       pas 70 ouverture vanne 3 L3
   // pas 80 demarrage rinçage                                      pas 90 fermeture vanne 3 L3                       pas 100 fermeture vanne 4 L2 et L3
   // pas 110 fermeture vanne station 1
   491: EQU(N7[105],10)XIC(N9[31].0)MOV(20,N7[105]);
   // pas 0 pas possible de démarrer la séquence             pas 5 pret                                                 pas 10 demarrage sequence ouverture vanne VA 1 de L3
   // pas 20 ouverutre vanne va1 station                        pas 30 fermeture vanne 2 L3                       pas 40 trnsfert naoh en cours attent arret
   // pas 50 ouverture vanne2 L3                                   pas 60 fermeture vanne 1 L3                       pas 70 ouverture vanne 3 L3
   // pas 80 demarrage rinçage                                      pas 90 fermeture vanne 3 L3                       pas 100 fermeture vanne 4 L2 et L3
   // pas 110 fermeture vanne station 1
   492: EQU(N7[105],20)XIC(N9[88].4)MOV(30,N7[105]);
   // pas 0 pas possible de démarrer la séquence             pas 5 pret                                                 pas 10 demarrage sequence ouverture vanne VA 1 de L3
   // pas 20 ouverutre vanne va1 station                        pas 30 fermeture vanne 2 L3                       pas 40 trnsfert naoh en cours attent arret
   // pas 50 ouverture vanne2 L3                                   pas 60 fermeture vanne 1 L3                       pas 70 ouverture vanne 3 L3
   // pas 80 demarrage rinçage                                      pas 90 fermeture vanne 3 L3                       pas 100 fermeture vanne 4 L2 et L3
   // pas 110 fermeture vanne station 1
   493: EQU(N7[105],30)XIC(N9[31].3)MOV(40,N7[105]);
   494: MOV(N9[106],N7[59]);
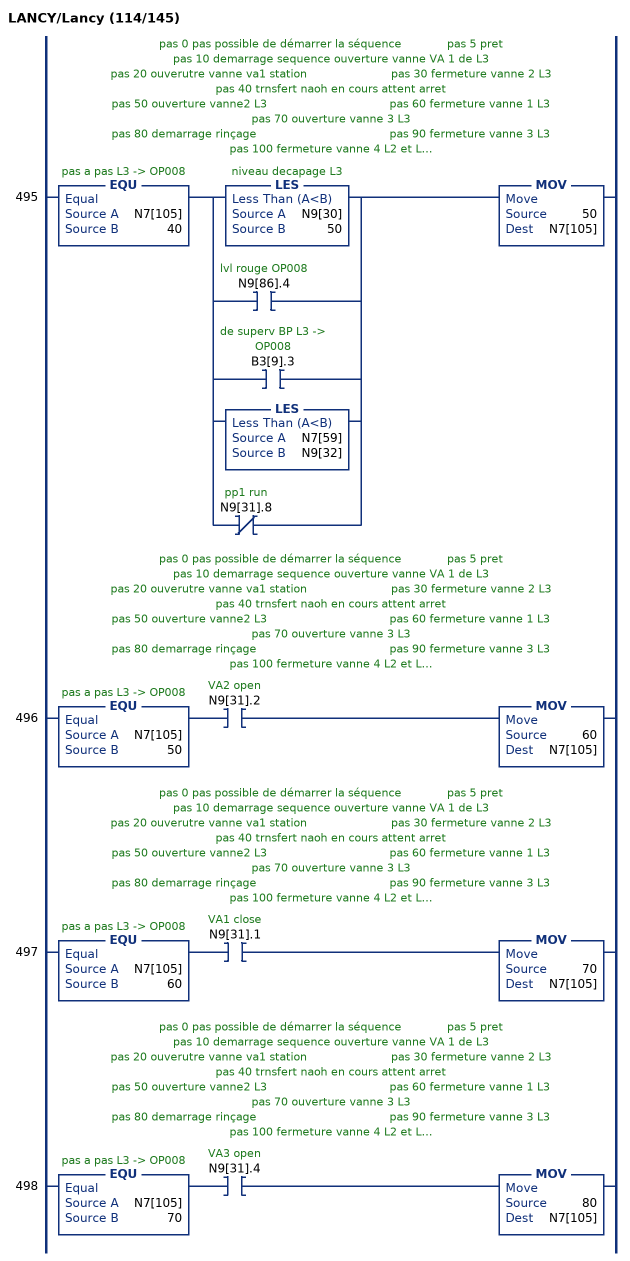
   // pas 0 pas possible de démarrer la séquence             pas 5 pret                                                 pas 10 demarrage sequence ouverture vanne VA 1 de L3
   // pas 20 ouverutre vanne va1 station                        pas 30 fermeture vanne 2 L3                       pas 40 trnsfert naoh en cours attent arret
   // pas 50 ouverture vanne2 L3                                   pas 60 fermeture vanne 1 L3                       pas 70 ouverture vanne 3 L3
   // pas 80 demarrage rinçage                                      pas 90 fermeture vanne 3 L3                       pas 100 fermeture vanne 4 L2 et L3
   // pas 110 fermeture vanne station 1
   495: EQU(N7[105],40)[LES(N9[30],50) ,XIC(N9[86].4) ,XIC(B3[9].3) ,LES(N7[59],N9[32]) ,XIO(N9[31].8) ]MOV(50,N7[105]);
   // pas 0 pas possible de démarrer la séquence             pas 5 pret                                                 pas 10 demarrage sequence ouverture vanne VA 1 de L3
   // pas 20 ouverutre vanne va1 station                        pas 30 fermeture vanne 2 L3                       pas 40 trnsfert naoh en cours attent arret
   // pas 50 ouverture vanne2 L3                                   pas 60 fermeture vanne 1 L3                       pas 70 ouverture vanne 3 L3
   // pas 80 demarrage rinçage                                      pas 90 fermeture vanne 3 L3                       pas 100 fermeture vanne 4 L2 et L3
   // pas 110 fermeture vanne station 1
   496: EQU(N7[105],50)XIC(N9[31].2)MOV(60,N7[105]);
   // pas 0 pas possible de démarrer la séquence             pas 5 pret                                                 pas 10 demarrage sequence ouverture vanne VA 1 de L3
   // pas 20 ouverutre vanne va1 station                        pas 30 fermeture vanne 2 L3                       pas 40 trnsfert naoh en cours attent arret
   // pas 50 ouverture vanne2 L3                                   pas 60 fermeture vanne 1 L3                       pas 70 ouverture vanne 3 L3
   // pas 80 demarrage rinçage                                      pas 90 fermeture vanne 3 L3                       pas 100 fermeture vanne 4 L2 et L3
   // pas 110 fermeture vanne station 1
   497: EQU(N7[105],60)XIC(N9[31].1)MOV(70,N7[105]);
   // pas 0 pas possible de démarrer la séquence             pas 5 pret                                                 pas 10 demarrage sequence ouverture vanne VA 1 de L3
   // pas 20 ouverutre vanne va1 station                        pas 30 fermeture vanne 2 L3                       pas 40 trnsfert naoh en cours attent arret
   // pas 50 ouverture vanne2 L3                                   pas 60 fermeture vanne 1 L3                       pas 70 ouverture vanne 3 L3
   // pas 80 demarrage rinçage                                      pas 90 fermeture vanne 3 L3                       pas 100 fermeture vanne 4 L2 et L3
   // pas 110 fermeture vanne station 1
   498: EQU(N7[105],70)XIC(N9[31].4)MOV(80,N7[105]);
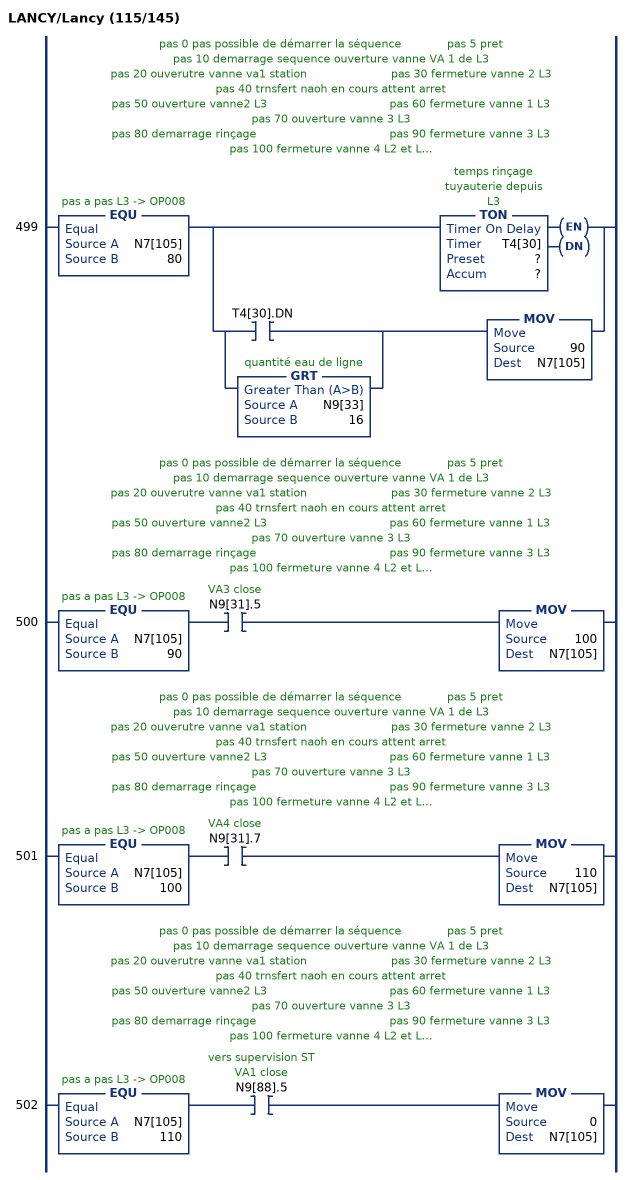
   // pas 0 pas possible de démarrer la séquence             pas 5 pret                                                 pas 10 demarrage sequence ouverture vanne VA 1 de L3
   // pas 20 ouverutre vanne va1 station                        pas 30 fermeture vanne 2 L3                       pas 40 trnsfert naoh en cours attent arret
   // pas 50 ouverture vanne2 L3                                   pas 60 fermeture vanne 1 L3                       pas 70 ouverture vanne 3 L3
   // pas 80 demarrage rinçage                                      pas 90 fermeture vanne 3 L3                       pas 100 fermeture vanne 4 L2 et L3
   // pas 110 fermeture vanne station 1
   499: EQU(N7[105],80)[TON(T4[30],?,?) ,[XIC(T4[30].DN) ,GRT(N9[33],16) ] MOV(90,N7[105]) ];
   // pas 0 pas possible de démarrer la séquence             pas 5 pret                                                 pas 10 demarrage sequence ouverture vanne VA 1 de L3
   // pas 20 ouverutre vanne va1 station                        pas 30 fermeture vanne 2 L3                       pas 40 trnsfert naoh en cours attent arret
   // pas 50 ouverture vanne2 L3                                   pas 60 fermeture vanne 1 L3                       pas 70 ouverture vanne 3 L3
   // pas 80 demarrage rinçage                                      pas 90 fermeture vanne 3 L3                       pas 100 fermeture vanne 4 L2 et L3
   // pas 110 fermeture vanne station 1
   500: EQU(N7[105],90)XIC(N9[31].5)MOV(100,N7[105]);
   // pas 0 pas possible de démarrer la séquence             pas 5 pret                                                 pas 10 demarrage sequence ouverture vanne VA 1 de L3
   // pas 20 ouverutre vanne va1 station                        pas 30 fermeture vanne 2 L3                       pas 40 trnsfert naoh en cours attent arret
   // pas 50 ouverture vanne2 L3                                   pas 60 fermeture vanne 1 L3                       pas 70 ouverture vanne 3 L3
   // pas 80 demarrage rinçage                                      pas 90 fermeture vanne 3 L3                       pas 100 fermeture vanne 4 L2 et L3
   // pas 110 fermeture vanne station 1
   501: EQU(N7[105],100)XIC(N9[31].7)MOV(110,N7[105]);
   // pas 0 pas possible de démarrer la séquence             pas 5 pret                                                 pas 10 demarrage sequence ouverture vanne VA 1 de L3
   // pas 20 ouverutre vanne va1 station                        pas 30 fermeture vanne 2 L3                       pas 40 trnsfert naoh en cours attent arret
   // pas 50 ouverture vanne2 L3                                   pas 60 fermeture vanne 1 L3                       pas 70 ouverture vanne 3 L3
   // pas 80 demarrage rinçage                                      pas 90 fermeture vanne 3 L3                       pas 100 fermeture vanne 4 L2 et L3
   // pas 110 fermeture vanne station 1
   502: EQU(N7[105],110)XIC(N9[88].5)MOV(0,N7[105]);
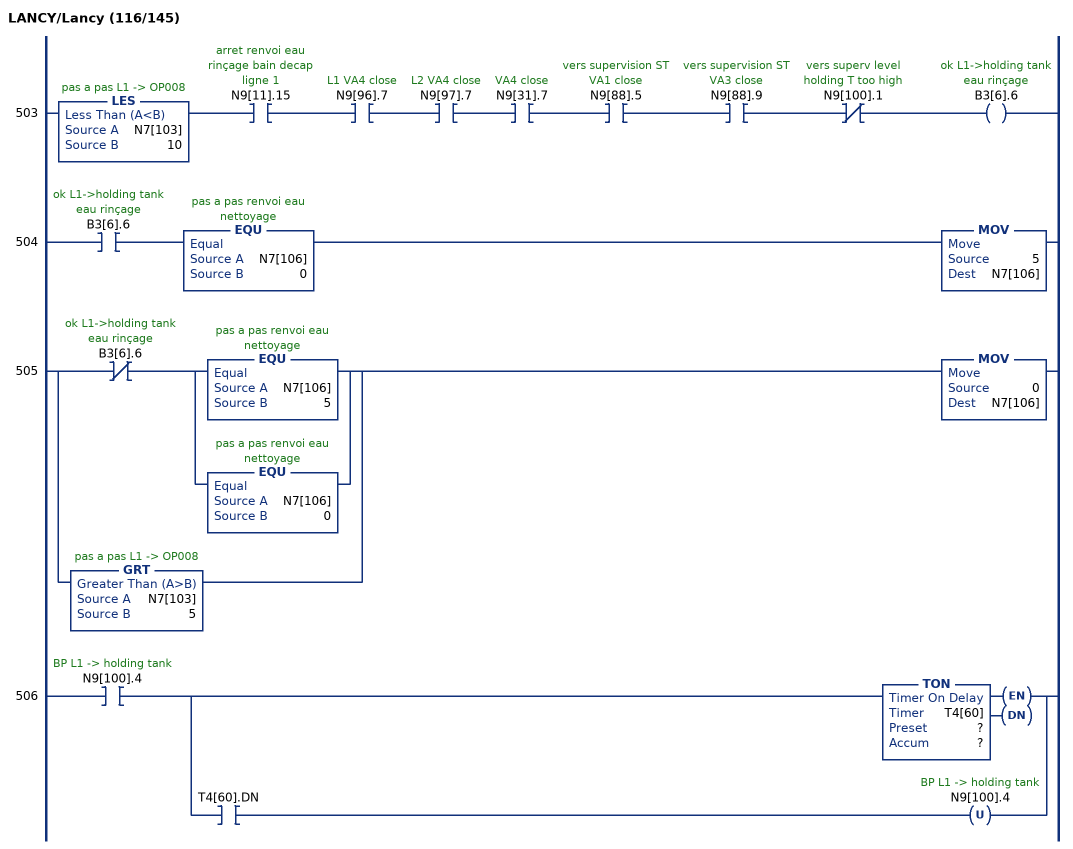
   503: LES(N7[103],10)XIC(N9[11].15)XIC(N9[96].7)XIC(N9[97].7)XIC(N9[31].7)XIC(N9[88].5)XIC(N9[88].9)XIO(N9[100].1)OTE(B3[6].6);
   504: XIC(B3[6].6)EQU(N7[106],0)MOV(5,N7[106]);
   505: [XIO(B3[6].6) [EQU(N7[106],5) ,EQU(N7[106],0) ] ,GRT(N7[103],5) ]MOV(0,N7[106]);
   506: XIC(N9[100].4)[TON(T4[60],?,?) ,XIC(T4[60].DN) OTU(N9[100].4) ];
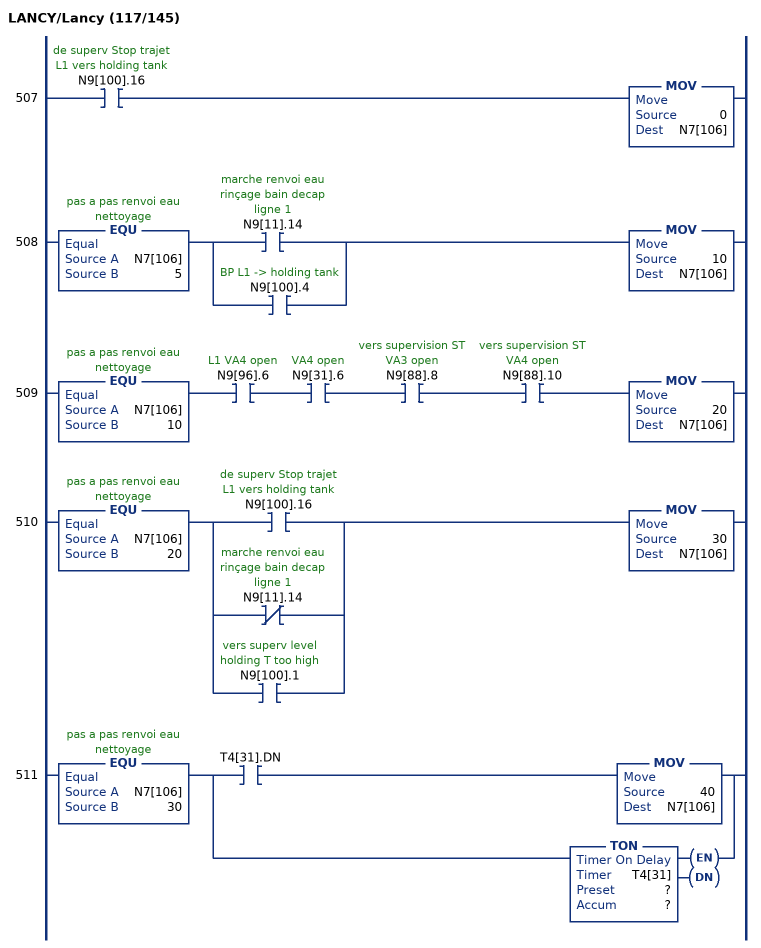
   507: XIC(N9[100].16)MOV(0,N7[106]);
   508: EQU(N7[106],5)[XIC(N9[11].14) ,XIC(N9[100].4) ]MOV(10,N7[106]);
   509: EQU(N7[106],10)XIC(N9[96].6)XIC(N9[31].6)XIC(N9[88].8)XIC(N9[88].10)MOV(20,N7[106]);
   510: EQU(N7[106],20)[XIC(N9[100].16) ,XIO(N9[11].14) ,XIC(N9[100].1) ]MOV(30,N7[106]);
   511: EQU(N7[106],30)[XIC(T4[31].DN) MOV(40,N7[106]) ,TON(T4[31],?,?) ];
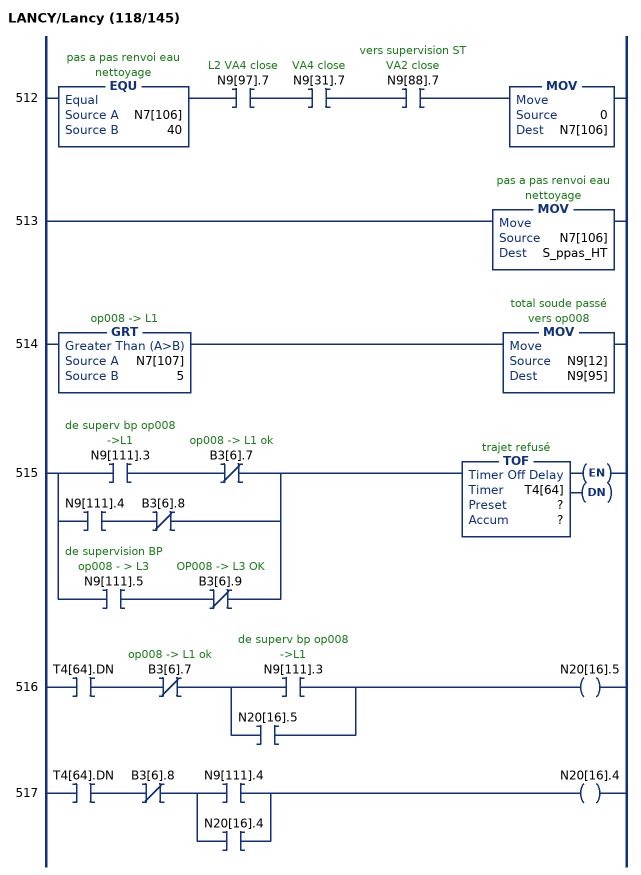
   512: EQU(N7[106],40)XIC(N9[97].7)XIC(N9[31].7)XIC(N9[88].7)MOV(0,N7[106]);
   513: MOV(N7[106],S_ppas_HT);
   514: GRT(N7[107],5)MOV(N9[12],N9[95]);
   515: [XIC(N9[111].3) XIO(B3[6].7) ,XIC(N9[111].4) XIO(B3[6].8) ,XIC(N9[111].5) XIO(B3[6].9) ]TOF(T4[64],?,?);
   516: XIC(T4[64].DN)XIO(B3[6].7)[XIC(N9[111].3) ,XIC(N20[16].5) ]OTE(N20[16].5);
   517: XIC(T4[64].DN)XIO(B3[6].8)[XIC(N9[111].4) ,XIC(N20[16].4) ]OTE(N20[16].4);
